PROGRAM ControlBox
VAR
	fbControlBox : FB_ControlBox; 
END_VAR

fbControlBox(
bRealControlBox := FALSE,
eMode => Work.eMode,
);

END_PROGRAM

(* stored: Version 1.1.0.1, ProductVersion 3.1.4024.9
   POU ControlBox: Id {f099b577-7c17-4f98-8e29-157282967496}, SpecialFunc None *)
